{attribute 'GeneratedUsingTerminal: EK1100-0000-0018'}
{attribute addProperty BoxType "EK1100-0000-0018"}
{attribute addProperty Id "Beckhoff_ATH2xxxEK1122Beckhoff_ATH2xxxEK1122_8B1D7AFC870A_0013_ATH2000_5250_0022ATH2000_37BB9B9414"}
{attribute addProperty CRC "2687039341"}
{attribute addProperty Size "884"}
TYPE Beckhoff_ATH2xxx_A028F76D EXTENDS EK1100_AB5A9467 :
STRUCT
	{attribute addProperty Name "Beckhoff_ATH2xxxEK1122"}
	Beckhoff_ATH2xxxEK1122 : Beckhoff_ATH2xxxEK1122_8B1D7AFC;
	{attribute addProperty Name "A_0013_ATH2000_5250_0022"}
	A_0013_ATH2000_5250_0022 : ATH2000_37BB9B94;
END_STRUCT
END_TYPE

(* stored: Version 1.2.0.0, ProductVersion 3.1.4024.9
   DUT Beckhoff_ATH2xxx_A028F76D: Id {33888f66-cac2-47e3-924a-e065e7ad2b3a} *)
